FUNCTION_BLOCK FB_XmlPersistentEventStorage IMPLEMENTS I_PersistentEventStorage
VAR_INPUT
END_VAR
VAR_OUTPUT
END_VAR
VAR
END_VAR


METHOD StoreEvent
VAR_INPUT
	stEvent	: ST_Event;
END_VAR
//  Here is the implementation of this method and XML writing is done to store the event
END_METHOD

END_FUNCTION_BLOCK

(* stored: Version 1.1.0.1, ProductVersion 3.1.4024.16
   POU FB_XmlPersistentEventStorage: Id {0f3984ac-7c24-4fdf-93c5-027661fcd10e}, SpecialFunc None
   Method StoreEvent: Id {acfa180f-3f4a-42fd-bc60-0a3c3f36290c} *)
